Fanuc KAREL source: kb00091.compact.KL

PROGRAM KB00091
%STACKSIZE=65535
%PRIORITY=65535
%NOLOCKGROUP
%ENVIRONMENT REGOPE
VAR
P1 : INTEGER
P2 : STRING[80]
P3 : INTEGER
BEGIN
P1=1
P2='A'
P3=1
GET_REG_CMT(P1,P2,P3)
END KB00091
